(* get pointer to axis data *)
pAxisData := gpAx[nHliAxIdx];
IF pAxisData^.ipo_state.cnc_channel_r = nChan THEN (* it's an axis of the channel *)
	(* is a reset commanded *)
	IF pAxisData^.ipo_lc_control.plc_reset.command_r = TRUE THEN
		(* quit this reset *)
		pAxisData^.ipo_lc_control.plc_reset.state_w := TRUE;

		ADSLOG2(strMsg:='Reset of axis: %d', nUDINT:=nAxisNr, strArg:='');

		HLI_AxisReset := TRUE;
	END_IF
END_IF

END_FUNCTION

// ---- POUs/CNC/F6 BlockSearch/HLI_ChannelBlockSearch.TcPOU
FUNCTION_BLOCK HLI_ChannelBlockSearch
VAR_INPUT
	nChan						: UDINT;			(* Number of channel *)
	(* interface values *)
	BlockSearch				: ST_BlockSearch;
END_VAR
VAR_IN_OUT
	bStartWrite				: BOOL;			(* Edge signal *)
	bStartRead				: BOOL;			(* Edge signal *)
END_VAR
VAR_OUTPUT
	Busy						: BOOL;
	Err						: BOOL;
	nErrorState				: UINT;
	(* interface values *)
	nActType					: INT;
	fActDistance			: LREAL;
	bActAutoReturn			: BOOL;
	nActDeviationMax		: UDINT;
	nActBlockNumber		: DINT;
	nActPass					: DINT;
	nActBlockCount			: DINT;
	(* current values *)
	actualBlockNumber		: DINT := 0;
	actualBlockCount		: DINT := 0;
	actualBlockCount_AferReset : DINT := 0;
	coveredDistance		: DINT;
END_VAR
VAR
	pChannel					: POINTER TO HIGH_LEVEL_INTERFACE_CH;
	nHliChIdx				: UDINT;
	bReadStarted			: BOOL;
	bWriteStarted			: BOOL;
	rtStartRead				: R_TRIG;
	rtStartWrite			: R_TRIG;

	fbWriteType				: FB_BlockSearchWrite;
	fbReadType				: FB_BlockSearchRead;

	fbWriteCovDistance	: FB_BlockSearchWrite;
	fbReadCovDistance		: FB_BlockSearchRead;

	fbWriteAutoReturn		: FB_BlockSearchWrite;
	fbReadAutoReturn		: FB_BlockSearchRead;

	fbWriteDeviationMax	: FB_BlockSearchWrite;
	fbReadDeviationMax	: FB_BlockSearchRead;

	fbWriteBlockNumber	: FB_BlockSearchWrite;
	fbReadBlockNumber		: FB_BlockSearchRead;
	fbReadActBlockNumber	: FB_BlockSearchRead;

	fbWriteBlockCount		: FB_BlockSearchWrite;
	fbReadBlockCount		: FB_BlockSearchRead;
	fbReadActBlockCount	: FB_BlockSearchRead;

	fbWritePass				: FB_BlockSearchWrite;
	fbReadPass				: FB_BlockSearchRead;

	nIdxGrp					: UDINT;
	fDist						: LREAL;
	timer1					: TON;				(* Timer to read actual values cyclically *)
	bStartReadAct			: BOOL;

	channelMode 			: DWORD;
	blockSearchStart		: BOOL;
END_VAR

(* ========================================================= *)
(*    FUN: HLI_ChannelBlockSearch                            *)
(* --------------------------------------------------------- *)
(*   Desc:                                                   *)
(* Author: MK                                                *)
(*   Date: 21.12.2011                                        *)
(*   Rev.: 1.0                                               *)
(* ========================================================= *)


nHliChIdx := nChan - 1;

IF nChan <= 0 OR gNrCh < nChan OR			(* check for channel no *)
	gpCh[nHliChIdx] = 0 THEN					(* check for zero pointer *)
	Err := TRUE;
	RETURN; (* e x i t *)
END_IF


pChannel := gpCh[nHliChIdx];
Err := FALSE;
nIdxGrp := 16#00020100 + nChan;
blockSearchStart := FALSE;


(* ----------------------------------- *)
(* --- write block search commands --- *)
(* ----------------------------------- *)

rtStartWrite(CLK:=bStartWrite);
IF rtStartWrite.Q THEN
	bWriteStarted := TRUE;
	bStartWrite := FALSE; (* reset the HMI signal *)
END_IF

IF bWriteStarted THEN
	Busy := TRUE;
	IF BlockSearch.nType = 5 THEN
		BlockSearch.nType := 3;								(* start position by block count *)

		BlockSearch.bAutoReturn := TRUE;
		(*nPass	:= 1;*)
	END_IF

	(* write block search data to Cnc *)
	fDist := BlockSearch.fDistance * 10.0;
	fbWriteType(nIdxGrp:=nIdxGrp, nIdxOffs:=16#49, nLen:=2, bStart:=rtStartWrite.Q, pDest:=ADR(BlockSearch.nType));
	fbWriteCovDistance(nIdxGrp:=nIdxGrp, nIdxOffs:=16#4A, nLen:=8, bStart:=rtStartWrite.Q, pDest:=ADR(fDist));
	fbWriteAutoReturn(nIdxGrp:=nIdxGrp, nIdxOffs:=16#4B, nLen:=1, bStart:=rtStartWrite.Q, pDest:=ADR(BlockSearch.bAutoReturn));
	fbWriteDeviationMax(nIdxGrp:=nIdxGrp, nIdxOffs:=16#4C, nLen:=4, bStart:=rtStartWrite.Q, pDest:=ADR(BlockSearch.nDeviationMax));
	fbWritePass(nIdxGrp:=nIdxGrp, nIdxOffs:=16#60, nLen:=4, bStart:=rtStartWrite.Q, pDest:=ADR(BlockSearch.nPass));

	CASE BlockSearch.nType OF		(* count and number share a part of the memory *)
		3:	fbWriteBlockCount(nIdxGrp:=nIdxGrp, nIdxOffs:=16#5E, nLen:=4, bStart:=rtStartWrite.Q, pDest:=ADR(BlockSearch.nBlockCount));
		4:	fbWriteBlockNumber(nIdxGrp:=nIdxGrp, nIdxOffs:=16#5F, nLen:=4, bStart:=rtStartWrite.Q, pDest:=ADR(BlockSearch.nBlockNumber));
	END_CASE

	IF fbWriteType.Busy = FALSE
		AND fbWriteCovDistance.BUSY = FALSE
		AND fbWriteAutoReturn.BUSY = FALSE
		AND fbWriteDeviationMax.BUSY = FALSE
		AND fbWriteBlockNumber.BUSY = FALSE
		AND fbWritePass.BUSY = FALSE
		AND fbWriteBlockCount.BUSY = FALSE
	THEN
		Busy := FALSE;
		bWriteStarted := FALSE;
		blockSearchStart := TRUE;
	END_IF
END_IF


(* Start block search *)
(*
IF (blockSearchStart) AND ((nType = 3) OR (nType = 4)) THEN
	PLCMachineMode[nChan].Start := TRUE;
END_IF
*)

(* -------------------------------- *)
(* --- read block search states --- *)
(* -------------------------------- *)

rtStartRead(CLK:=bStartRead);
(*rtStartRead(CLK:=Timer.Q);*)
IF rtStartRead.Q THEN
	bReadStarted := TRUE;
END_IF

IF bReadStarted THEN
	Busy := TRUE;

	fbReadType(nIdxGrp:=nIdxGrp, nIdxOffs:=16#61, nLen:=2, bStart:=rtStartRead.Q, pDest:=ADR(nActType));
	fbReadCovDistance(nIdxGrp:=nIdxGrp, nIdxOffs:=16#62, nLen:=8, bStart:=rtStartRead.Q, pDest:=ADR(fActDistance));
	fbReadAutoReturn(nIdxGrp:=nIdxGrp, nIdxOffs:=16#63, nLen:=1, bStart:=rtStartRead.Q, pDest:=ADR(bActAutoReturn));
	fbReadDeviationMax(nIdxGrp:=nIdxGrp, nIdxOffs:=16#64, nLen:=4, bStart:=rtStartRead.Q, pDest:=ADR(nActDeviationMax));
	CASE nActType OF			(* count and number cannot be read within a single cycle! *)
		3: fbReadBlockCount(nIdxGrp:=nIdxGrp, nIdxOffs:=16#76, nLen:=4, bStart:=rtStartRead.Q, pDest:=ADR(nActBlockCount));
		4: fbReadBlockNumber(nIdxGrp:=nIdxGrp, nIdxOffs:=16#77, nLen:=4, bStart:=rtStartRead.Q, pDest:=ADR(nActBlockNumber));
	END_CASE;
	fbReadPass(nIdxGrp:=nIdxGrp, nIdxOffs:=16#78, nLen:=4, bStart:=rtStartRead.Q, pDest:=ADR(nActPass));

	(*
	fbReadActBlockNumber(nIdxGrp:=nIdxGrp, bStart:=rtStartRead.Q, pDest:=ADR(actualBlockNumber));
	fbReadActBlockCount(nIdxGrp:=nIdxGrp, bStart:=rtStartRead.Q, pDest:=ADR(actualBlockCount));
	*)

	IF fbReadType.Busy = FALSE
		AND fbReadCovDistance.Busy = FALSE
		AND fbReadAutoReturn.Busy = FALSE
		AND fbReadDeviationMax.Busy = FALSE
		AND fbReadBlockNumber.Busy = FALSE
		AND fbReadPass.Busy = FALSE
		AND fbReadActBlockNumber.Busy = FALSE
		AND fbReadActBlockCount.Busy = FALSE
	THEN
		Busy := FALSE;

		bReadStarted := FALSE;
		bStartRead := FALSE; (* reset the HMI signal *)
	END_IF
END_IF


(* Start a cyclic timer with period 100 ms *)
timer1(IN := NOT(timer1.Q), PT := T#100MS);
IF timer1.Q THEN
	bStartReadAct := TRUE;
END_IF

IF bStartReadAct THEN
	fbReadActBlockNumber(nIdxGrp:=nIdxGrp, nIdxOffs:=16#0E, nLen:=4, bStart:=TRUE, pDest:=ADR(actualBlockNumber));
	fbReadActBlockCount(nIdxGrp:=nIdxGrp, nIdxOffs:=16#0D, nLen:=4, bStart:=TRUE, pDest:=ADR(actualBlockCount));
	
	IF fbReadActBlockNumber.Busy = FALSE
		AND fbReadActBlockNumber.Busy = FALSE
	THEN
		bStartReadAct := FALSE;
	END_IF
END_IF


(* just read actual covered distance *)
coveredDistance := pChannel^.bahn_state.covered_distance_r;

(* save all the information from the Cnc break *)
channelMode := HLI_ChannelGetMode(nChan);
IF (actualBlockCount <> 0) AND (channelMode = HLI_IMCM_AUTOMATIC_MODE) THEN
	(* Information stayes after reset *)
	actualBlockCount_AferReset := actualBlockCount;
END_IF


(*actualBlockNumber := pglAx[0]^.lr_state.block_nr_r;  asume first axis is always moved *)


(* handshake during block search on/off *)
pChannel^.bahn_lc_control.block_search.enable_w := TRUE;

IF pChannel^.bahn_lc_control.block_search.command_r <>
	pChannel^.bahn_lc_control.block_search.state_w THEN

	(* acknowledge *)
	pChannel^.bahn_lc_control.block_search.state_w := pChannel^.bahn_lc_control.block_search.command_r;

(*
	(* pup up of change *)
	IF pChannel^.bahn_lc_control.block_search.state_w THEN
		ADSLOGDINT( msgCtrlMask := ADSLOG_MSGTYPE_MSGBOX OR ADSLOG_MSGTYPE_LOG,
						msgFmtStr := 'block search: %d', dintArg := 1);
	ELSE
		ADSLOGDINT( msgCtrlMask := ADSLOG_MSGTYPE_MSGBOX OR ADSLOG_MSGTYPE_LOG,
						msgFmtStr := 'block search: %d', dintArg := 0);
	END_IF
*)
END_IF

END_FUNCTION_BLOCK

// ---- POUs/CNC/F6 BlockSearch/FB_BlockSearchWrite.TcPOU
FUNCTION_BLOCK FB_BlockSearchWrite
VAR_INPUT
	nIdxGrp					: UDINT;
	nIdxOffs					: UDINT;
	nLen						: UDINT;
	bStart					: BOOL;
	pDest						: POINTER TO DWORD;
END_VAR
VAR_OUTPUT
	Busy						: BOOL;
	bErr						: BOOL;
END_VAR
VAR
   fbWrite              : ADSWRITE;
   bStarted             : BOOL;
END_VAR

IF bStarted = FALSE THEN
   IF bStart = TRUE THEN
      bStarted := TRUE;
      bErr := FALSE;
      Busy := TRUE;
   END_IF
END_IF

IF bStarted THEN
   (* raising edge of Timer triggers write request *)
   fbWrite(NetID:='', Port:=553, IdxGrp:=nIdxGrp, IdxOffs:=nIdxOffs,
         LEN:=nLen, SrcAddr:=pDest, WRITE:=bStarted, TMOUT:=T#1S);
   IF NOT fbWrite.Busy THEN
      (* There was an error in the execution of the write request *)
      IF fbWrite.Err THEN
         bErr := TRUE;
      END_IF
      fbWrite(WRITE := FALSE);    (* reset because of edge detection in FB ADSWRITE *)
      bStarted := FALSE;
      Busy := FALSE;
   END_IF
END_IF

END_FUNCTION_BLOCK

// ---- POUs/CNC/F6 BlockSearch/FB_BlockSearchRead.TcPOU
FUNCTION_BLOCK FB_BlockSearchRead
VAR_INPUT
	nIdxGrp					: UDINT;
	nIdxOffs					: UDINT;
	nLen						: UDINT;
	bStart					: BOOL;
	pDest						: POINTER TO DWORD;
END_VAR
VAR_OUTPUT
	Busy						: BOOL;
	bErr						: BOOL;
END_VAR
VAR
	fbRead					: ADSREAD;
	bStarted					: BOOL;
END_VAR

IF bStarted = FALSE THEN
	IF bStart = TRUE THEN
		bStarted := TRUE;
		bErr := FALSE;
		Busy := TRUE;
	END_IF
END_IF

IF bStarted THEN
	(* raising edge of Timer triggers read request *)
	fbRead(NetID:='', Port:=553, IdxGrp:=nIdxGrp, IdxOffs:=nIdxOffs,
		LEN:=nLen, DestAddr:=pDest, READ:=bStarted, TMOUT:=T#1S);
	IF NOT fbRead.Busy THEN
		(* There was an error in the execution of the read request *)
		IF fbRead.Err THEN
			bErr := TRUE;
		END_IF
		fbRead(READ := FALSE);    (* reset because of edge detection in FB ADSREAD *)
		bStarted := FALSE;
		Busy := FALSE;
	END_IF
END_IF

END_FUNCTION_BLOCK

// ---- POUs/CNC/F3_Control/HLI_ChannelGetMessage.TcPOU
FUNCTION_BLOCK HLI_ChannelGetMessage
VAR_INPUT
	nChan			: UINT;			(* Number of channel *)
	bExecute  	: BOOL := FALSE;
	bShowDlg		: BOOL := FALSE;
END_VAR
VAR_OUTPUT
	strToPLC		: STRING(HLI_MSG_CONTENT_STRL) := '';
	iMsgType		: DWORD := 0;
END_VAR
VAR
	nHliChIdx	: UINT;
	pChannel		: POINTER TO HIGH_LEVEL_INTERFACE_CH;
	pMsgCU		: POINTER TO MC_CONTROL_MSG_UNIT;
	pMsgToPLC	: POINTER TO STRING(HLI_MSG_CONTENT_STRL);
END_VAR

(* ========================================================= *)
(*     FB: HLI_ChannelGetMessage                             *)
(* --------------------------------------------------------- *)
(*   Desc: Get message from the CNC                          *)
(*   Author: MK                                              *)
(*   Date: 16.11.2006                                        *)
(*   Rev.: 1.00                                              *)
(* ========================================================= *)


nHliChIdx := nChan - 1;

IF nChan <= 0 OR gNrCh < nChan OR			(* check for channel no *)
	gpCh[nHliChIdx] = 0 THEN					(* check for zero pointer *)
	RETURN; (* e x i t *)
END_IF

IF bExecute = FALSE THEN
	RETURN; (* e x i t *)
END_IF

(* Get pointer to data of a specific channel at the HLI *)
pChannel := gpCh[nHliChIdx];

(* Control unit at the HLI that handles channel specific messages *)
pMsgCU := ADR(pChannel^.msg_mc_control);

(* Is the complete message in the control unit? *)
IF pMsgCU^.request_semaphor_rw = TRUE THEN
	(* Pointer to content of the message sent to the PLC *)
	pMsgToPLC := ADR(pMsgCU^.request_r.inhalt);

	(* Get the message from the control unit *)
	strToPLC := pMsgToPLC^;

	CncSystem.Channel[nChan].Message := strToPLC;
	
	(* Get the message type *)
	iMsgType := pMsgCU^.request_r.typ;

	(* Pop up dialog with the message send to the PLC *)
	IF bShowDlg THEN
		ADSLOGSTR( msgCtrlMask :=ADSLOG_MSGTYPE_MSGBOX OR ADSLOG_MSGTYPE_LOG,
						msgFmtStr := 'Message sent to PLC via HLI:%s',
						strArg := strToPLC);
	END_IF

	(* Acknowledge that you got the message *)
	pChannel^.msg_mc_control.request_semaphor_rw  := FALSE;
END_IF

END_FUNCTION_BLOCK

// ---- POUs/CncAxisEnable.TcPOU
PROGRAM CncAxisEnable
VAR_INPUT
	bEnable					: BOOL;
END_VAR
VAR
	bTorquePermission		: BOOL;
	bFeedhold				: BOOL;
	bDriveOn					: BOOL;

	T_DriveOn				: TON;
END_VAR

(* ========================================================= *)
(*    PRG: CncAxisEnable                                     *)
(* --------------------------------------------------------- *)
(*   Desc:                                                   *)
(* Author: MK                                                *)
(*   Date: 21.12.2011                                        *)
(*   Rev.: 1.0                                               *)
(* ========================================================= *)


(* Enable drive, order depends by type of drive and fieldbus *)
T_DriveOn(IN:=bEnable, PT:=T#1S);
IF bEnable THEN
	bDriveOn			:= TRUE;
	IF T_DriveOn.Q THEN
		bTorquePermission	:= TRUE;
		bFeedhold			:= TRUE;
	END_IF
ELSE
	bTorquePermission	:= FALSE;
	bFeedhold			:= FALSE;
	bDriveOn				:= FALSE;
END_IF

(* Enable drive, order depends by type of drive and fieldbus *)
(*
T_DriveOn(IN:=bEnable, PT:=T#1s);
IF bEnable THEN
	bTorquePermission	:= TRUE;
	bFeedhold			:= TRUE;
	IF T_DriveOn.Q THEN
		bDriveOn			:= TRUE;
	END_IF
ELSE
	bTorquePermission	:= FALSE;
	bFeedhold			:= FALSE;
	bDriveOn				:= FALSE;
END_IF
*)


(* Controller Enable, axis specific *)
HLI_AxisSetFeedHold(Axis:=1, TorquePermission:=bTorquePermission, Feedhold:=bFeedhold, DriveOn:=bDriveOn);
HLI_AxisSetFeedHold(Axis:=2, TorquePermission:=bTorquePermission, Feedhold:=bFeedhold, DriveOn:=bDriveOn);
HLI_AxisSetFeedHold(Axis:=3, TorquePermission:=bTorquePermission, Feedhold:=bFeedhold, DriveOn:=bDriveOn);
HLI_AxisSetFeedHold(Axis:=4, TorquePermission:=bTorquePermission, Feedhold:=bFeedhold, DriveOn:=bDriveOn);
HLI_AxisSetFeedHold(Axis:=5, TorquePermission:=bTorquePermission, Feedhold:=bFeedhold, DriveOn:=bDriveOn);

HLI_AxisSetFeedHold(Axis:=6, TorquePermission:=bTorquePermission, Feedhold:=bFeedhold, DriveOn:=bDriveOn);
HLI_AxisSetFeedHold(Axis:=7, TorquePermission:=bTorquePermission, Feedhold:=bFeedhold, DriveOn:=bDriveOn);
HLI_AxisSetFeedHold(Axis:=8, TorquePermission:=bTorquePermission, Feedhold:=bFeedhold, DriveOn:=bDriveOn);

END_PROGRAM

// ---- POUs/CNC/F3_Control/HLI_AxisSetFeedHold.TcPOU
FUNCTION HLI_AxisSetFeedHold : BOOL
VAR_INPUT
	Axis					: UDINT;
	TorquePermission	: BOOL;
	Feedhold				: BOOL;
	DriveOn				: BOOL;
END_VAR
VAR
	nHliAxIdx			: UDINT;		(* Index of axis specific HLI area *)
END_VAR

(* ========================================================= *)
(*    FUN: HLI_AxisSetFeedHold                               *)
(* --------------------------------------------------------- *)
(*   Desc:                                                   *)
(* Author: MK                                                *)
(*   Date: 21.12.2011                                        *)
(*   Rev.: 1.0                                               *)
(* ========================================================= *)


nHliAxIdx := Axis - 1;

IF Axis < 1	OR gNrAx < Axis			(* check for axis no *)
	OR gpAx[nHliAxIdx] = 0 THEN		(* check for zero pointer *)
	HLI_AxisSetFeedHold := FALSE;
	RETURN; (* e x i t *)
END_IF

(* set regulation and feed *)
gpAx[nHliAxIdx]^.lr_mc_control.torque_permission.command_w := TorquePermission;
gpAx[nHliAxIdx]^.lr_mc_control.release_feedhold.command_w := Feedhold;
gpAx[nHliAxIdx]^.lr_mc_control.drive_on.command_w := DriveOn;

HLI_AxisSetFeedHold := TRUE;

END_FUNCTION

// ---- POUs/CNC/F3_Control/HLI_AxisSetTrackingOperation.TcPOU
FUNCTION HLI_AxisSetTrackingOperation : BOOL
VAR_INPUT
	nAxisNr				: UDINT;
	bPLCAxisEnable    : BOOL;
END_VAR
VAR
	nHliAxIdx			: UDINT;		(* Index of axis specific HLI area *)
END_VAR

(* ========================================================= *)
(*    FUN: HLI_AxisSetTrackingOperation                      *)
(* --------------------------------------------------------- *)
(*   Desc:                                                   *)
(*   Author: TV                                              *)
(*   Date: 21.12.2012                                        *)
(*   Rev.: 1.0                                               *)
(* ========================================================= *)


nHliAxIdx := nAxisNr - 1;

IF nAxisNr < 1	OR gNrAx < nAxisNr	(* check for axis no *)
	OR gpAx[nHliAxIdx] = 0 THEN		(* check for zero pointer *)
	HLI_AxisSetTrackingOperation := FALSE;
	RETURN; (* e x i t *)
END_IF


(* The axis is set to tracking operation (follow up) on or off, i.e. the control loop is opened.
   The command position implicitly is set to the actual position. *)
IF gpAx[nHliAxIdx]^.lr_state.axis_state_r = HLI_AXIS_ERROR OR NOT bPLCAxisEnable THEN
	gpAx[nHliAxIdx]^.lr_mc_control.follow_up.command_w := TRUE;
	HLI_AxisSetTrackingOperation := TRUE;
ELSE
	gpAx[nHliAxIdx]^.lr_mc_control.follow_up.command_w := FALSE;
	HLI_AxisSetTrackingOperation := FALSE;
END_IF

END_FUNCTION

// ---- POUs/CNC/F3_Control/HLI_AxisSetReferenceCam.TcPOU
FUNCTION HLI_AxisSetReferenceCam : BOOL
VAR_INPUT
	Axis					: UDINT;
	bReferenceCam		: BOOL;
END_VAR
VAR
	nHliAxIdx			: UDINT;		(* Index of axis specific HLI area *)
END_VAR

(* ========================================================= *)
(*    FUN: HLI_AxisSetReferenceCam                           *)
(* --------------------------------------------------------- *)
(*   Desc:                                                   *)
(* Author: MK                                                *)
(*   Date: 21.12.2011                                        *)
(*   Rev.: 1.0                                               *)
(* ========================================================= *)


nHliAxIdx := Axis - 1;

IF Axis < 1	OR gNrAx < Axis				(* check for axis no *)
	OR gpAx[nHliAxIdx] = 0 THEN			(* check for zero pointer *)
	HLI_AxisSetReferenceCam := FALSE;
	RETURN; (* e x i t *)
END_IF

(* set reference cam *)
gpAx[nHliAxIdx]^.lr_mc_control.reference_cam.command_w := bReferenceCam;

HLI_AxisSetReferenceCam := TRUE;

END_FUNCTION

// ---- POUs/CNC/F3_Control/HLI_ChannelSetOverride.TcPOU
FUNCTION HLI_ChannelSetOverride : BOOL
VAR_INPUT
	nChan					: UINT;			(* Number of channel *)
	nOverride			: UINT;
END_VAR
VAR
	nHliChIdx			: UINT;
END_VAR

(* ========================================================= *)
(*    FUN: HLI_ChannelSetOverride                            *)
(* --------------------------------------------------------- *)
(*   Desc: Set the channel Override                          *)
(* Author: MK                                                *)
(*   Date: 21.12.2011                                        *)
(*   Rev.: 1.0                                               *)
(* ========================================================= *)


nHliChIdx := nChan - 1;

IF nChan <= 0 OR gNrCh < nChan OR			(* check for channel no *)
	gpCh[nHliChIdx] = 0 THEN					(* check for zero pointer *)
	HLI_ChannelSetOverride := FALSE;
	RETURN; (* e x i t *)
END_IF

(* Limit the override *)
IF nOverride > 1200	THEN nOverride := 1200; END_IF
IF nOverride < 0 THEN nOverride := 0; END_IF

gpCh[nHliChIdx]^.bahn_mc_control.override_feedrate.command_w := nOverride;

HLI_ChannelSetOverride := TRUE;

END_FUNCTION

// ---- POUs/CNC/F3_Control/HLI_ChannelSetSuspendAxisOutput.TcPOU
FUNCTION HLI_ChannelSetSuspendAxisOutput : BOOL
VAR_INPUT
	nChan					: UDINT;			(* Number of channel *)
	bSuspendAxis		: BOOL;
END_VAR
VAR
	nHliChIdx			: UDINT;
END_VAR

(* ========================================================= *)
(*    FUN: HLI_ChannelSuspendAxisOutput                      *)
(* --------------------------------------------------------- *)
(*   Desc:                                                   *)
(* Author: MK                                                *)
(*   Date: 18.04.2003                                        *)
(*   Rev.: 1.0                                               *)
(* ========================================================= *)


nHliChIdx := nChan - 1;

IF nChan <= 0 OR gNrCh < nChan OR			(* check for channel no *)
	gpCh[nHliChIdx] = 0 THEN					(* check for zero pointer *)
	HLI_ChannelSetSuspendAxisOutput := FALSE;
	RETURN; (* e x i t *)
END_IF

gpCh[nHliChIdx]^.bahn_mc_control.suspend_axis_output.command_w := bSuspendAxis;

HLI_ChannelSetSuspendAxisOutput := TRUE;

END_FUNCTION

// ---- POUs/CNC/F9_Misc/HandWheel/PRG_ManualModeG201.TcPOU
PROGRAM PRG_ManualModeG201
VAR_INPUT
	nChan						: UDINT;		(* starts with 1, 2,... *)
END_VAR
VAR
	nAxis						: UINT := 3;	(* X=1; Y=2; Z=3 *)
	bOpModeAuto				: BOOL;		(* activates, deactivates operation *) 
	bManualIsOn				: BOOL;
	bEndOfManualMode		: BOOL;
	bManualModeErr			: BOOL;		(* inicates error *)

	AxisManualModeG201	: HLI_AxisManualMode;
	manualModeParam		: ST_ManualModeParam;
	pChannel					: POINTER TO HIGH_LEVEL_INTERFACE_CH;  		
	nHliChIdx				: UDINT;
	fbRTrig					: R_TRIG;
	fbFTrig					: F_TRIG;
	hbStateAxis				: DINT;
END_VAR

(* ========================================================= *)
(*    PRG: PRG_ManualModeG201                                *)
(* --------------------------------------------------------- *)
(*   Desc: Axis manual mode with parallel interpolation G201 *)
(* Author: MK                                                *)
(*   Date: 12.05.2016                                        *)
(*   Rev.: 1.0                                               *)
(* ========================================================= *)


nHliChIdx := nChan - 1;

IF nChan <= 0 OR gNrCh < nChan OR			(* check for channel no *)
	gpCh[nHliChIdx] = 0 THEN					(* check for zero pointer *)
	RETURN; (* e x i t *)
END_IF

(* axis number must be 1, 2, 3,... *)
IF nAxis < 1 THEN
	RETURN;
END_IF

(* activates operation only in automatic mode *)
bOpModeAuto := (HLI_ChannelGetMode(nChan:=nChan) = HLI_IMCM_AUTOMATIC_MODE);

(* This enables automatically the axis manual movement *)
pChannel := gpCh[nHliChIdx];
hbStateAxis := pChannel^.bahn_state.coord_r[nAxis - 1].hb_display_r.state;	(* Status of the axis | 0=Inactive, 1=Ready, 2=Active *)

fbRTrig(CLK := (hbStateAxis<>0) AND bOpModeAuto);
fbFTrig(CLK := (hbStateAxis<>0) AND bOpModeAuto);

IF fbRTrig.Q OR bManualIsOn THEN
	IF fbRTrig.Q THEN			(* activation *)
		bManualIsOn := TRUE;
		bEndOfManualMode := FALSE;
	ELSIF fbFTrig.Q THEN		(* deactivation *)
		bEndOfManualMode := TRUE;
	END_IF
	
	manualModeParam.nOpMode := UDINT_TO_UINT(HLI_HB_MODE_HR);
	manualModeParam.nLogAxisNr := nAxis;		// PlcManualModeSelectedAxis;
	manualModeParam.nControlElement := 1;
	manualModeParam.nHandwheelNr := 0;
	manualModeParam.nHandwheelIncs := PlcManualModeHandWheelIncs;
	manualModeParam.nHandwheelRes := PlcManualModeHandWheelRes; 
	manualModeParam.nTipSpeed := PlcManualModeSpeed;
	manualModeParam.nJogSpeed := PlcManualModeSpeed;
	manualModeParam.nJogDistance := PlcManualModeIncrements;

	(* manual mode keypress *)
	manualModeParam.bKeyPos := PlcManualModeRightKey;
	manualModeParam.bKeyNeg := PlcManualModeLeftKey;
	manualModeParam.bKeyRapid := PlcManualModeRapidFeedKey;

	
	AxisManualModeG201(nChan			:= nChan,
							sProgramName	:= '',
							bEndManual		:= bEndOfManualMode,
							ManualModeParam:= manualModeParam, 
							nKeyUnitIdx		:= 0,
							bManualModeHMI	:= FALSE,
							bReset			:= FALSE,
							bG201				:= TRUE);
							
	IF AxisManualModeG201.Busy = FALSE THEN
		AxisManualModeG201.bG201 := FALSE;
		bEndOfManualMode := FALSE;
		bManualIsOn := FALSE;
	END_IF
	bManualModeErr := AxisManualModeG201.Err;
END_IF

END_PROGRAM

// ---- POUs/CncMFunctions.TcPOU
PROGRAM CncMFunctions
VAR

END_VAR

(* ========================================================= *)
(*    FUN: CncMFunctions                                     *)
(* --------------------------------------------------------- *)
(*   Desc:                                                   *)
(* Author: MK                                                *)
(*   Date: 21.12.2011                                        *)
(*   Rev.: 1.0                                               *)
(* ========================================================= *)

(*
IF CncSystem.Channel[1].M[40] = TRUE THEN
	CncSystem.Channel[1].M[40] := FALSE;
END_IF
*)

(* M-functions *)
IF CNCSystem.Channel[1].M[17] = TRUE THEN
	CNCSystem.Channel[1].M[17] := FALSE;
END_IF

(*IF CNCSystem.Channel[1].M[52] = TRUE THEN
	Temp_Tabuleiro_set:=CNCSystem.Channel[1].M_Argument[52];
		IF (IOs.Temp_Tabuleiro<Temp_Tabuleiro_set+100 AND IOs.Temp_Tabuleiro>Temp_Tabuleiro_set-100) OR Temp_Tabuleiro_set=0 THEN
			CNCSystem.Channel[1].M[52] := FALSE;
		END_IF
END_IF*)

END_PROGRAM

// ---- POUs/CncPlcManualFunctions.TcPOU
PROGRAM CncPlcManualFunctions
VAR
	bSetString					: BOOL := TRUE;
	PLCManual_Off				: BYTE := 0;
	PLCManual_StatusLeft		: BYTE := 1;
	PLCManual_StatusRight	: BYTE := 2;
	PLCManual_LockLeft		: BYTE := 32;
	PLCManual_LockRight		: BYTE := 64;
END_VAR

(* ========================================================= *)
(*    FUN: CncPlcManualFunctions                             *)
(* --------------------------------------------------------- *)
(*   Desc:                                                   *)
(* Author: MK                                                *)
(*   Date: 21.08.2008                                        *)
(*   Rev.: 1.0                                               *)
(* ========================================================= *)


(* Manual functions *)
PortalStatus[1] := PLCManual_StatusLeft;
PortalStatus[2] := PLCManual_StatusLeft;
PortalStatus[3] := PLCManual_StatusLeft;
PortalStatus[4] := PLCManual_LockRight;

SchweissenStatus[1] := PLCManual_Off;
SchweissenStatus[2] := PLCManual_StatusLeft;
SchweissenStatus[3] := PLCManual_StatusRight;
SchweissenStatus[4] := PLCManual_StatusLeft;

MSGList3[3] := PortalOn[7];


IF bSetString THEN
	PortalActValueLeft[3] := INT_TO_STRING(DemoUpDown.UpDown);
	PortalActValueLeft[4] := INT_TO_STRING(DemoUpDown.UpDown);
	PortalActValueLeft[5] := INT_TO_STRING(DemoUpDown.UpDown);
END_IF

END_PROGRAM

// ---- POUs/CncPlcMessages.TcPOU
PROGRAM CncPlcMessages
VAR
	bShowMessage		: BOOL;
	
	event1				: FB_SimpleAdsLogEvent;
	event2				: FB_SimpleAdsLogEvent;
	bStartEvent			: BOOL;
	bStartEvent2		: BOOL;
	i						: INT;
END_VAR

(* ========================================================= *)
(*    FUN: CncPlcMessages                                    *)
(* --------------------------------------------------------- *)
(*   Desc:                                                   *)
(* Author: MK                                                *)
(*   Date: 21.12.2011                                        *)
(*   Rev.: 1.0                                               *)
(* ========================================================= *)


(* Messages *)
MSGList1[5] := bShowMessage;
MSGList1[6] := bShowMessage;
MSGList1[7] := bShowMessage;

(*FOR i:=1 TO 50 DO
	MSGList2[i] := bShowMessage;
END_FOR*)


// Eventlogger
(*
event1(SourceID:=50, EventID:=3, bSetEvent:=bStartEvent);
errId := event1.ErrId;

event2(SourceID:=50, EventID:=4, bSetEvent:=bStartEvent2);
*)

END_PROGRAM

// ---- POUs/CncRefPosOffs.TcPOU
PROGRAM CncRefPosOffs
VAR
END_VAR

(* ========================================================= *)
(*    FUN: CncRefPosOffs                                     *)
(* --------------------------------------------------------- *)
(*   Desc:                                                   *)
(* Author: MK                                                *)
(*   Date: 21.12.2011                                        *)
(*   Rev.: 1.0                                               *)
(* ========================================================= *)


gpAx[0]^.lr_mc_control.refpos_position.enable_w := TRUE;
gpAx[1]^.lr_mc_control.refpos_position.enable_w := TRUE;
gpAx[2]^.lr_mc_control.refpos_position.enable_w := TRUE;

gpAx[0]^.lr_mc_control.set_reference_position.enable_w := TRUE;  
gpAx[1]^.lr_mc_control.set_reference_position.enable_w := TRUE;  
gpAx[2]^.lr_mc_control.set_reference_position.enable_w := TRUE;  



gpAx[0]^.lr_mc_control.refpos_position.command_w := 100 * 10000;
gpAx[1]^.lr_mc_control.refpos_position.command_w := 200 * 10000;
gpAx[2]^.lr_mc_control.refpos_position.command_w := 300 * 10000;

gpAx[0]^.lr_mc_control.set_reference_position.command_w := TRUE;  
gpAx[1]^.lr_mc_control.set_reference_position.command_w := TRUE;  
gpAx[2]^.lr_mc_control.set_reference_position.command_w := TRUE;

END_PROGRAM

// ---- POUs/CncVariables.TcPOU
PROGRAM CncVariables
VAR_INPUT
END_VAR
VAR
	VE						: ST_VEVariableConfig;
	v1 : DINT;
	v4 : DINT;
	v5 : DINT;
END_VAR

(* ========================================================= *)
(*    PRG: CncVariables                                      *)
(* --------------------------------------------------------- *)
(*   Desc:                                                   *)
(* Author: MK                                                *)
(*   Date: 21.12.2011                                        *)
(*   Rev.: 1.0                                               *)
(* ========================================================= *)



(* External Variables in the CNC, must be set only at startup *)
VE.VARIABLE_1 := LinkVEChannelStructure(nChan:=1, nVEIndex:=0, bGlobal:=TRUE);
VE.VARIABLE_4 := LinkVEChannelStructure(nChan:=1, nVEIndex:=3, bGlobal:=TRUE);
VE.VARIABLE_5 := LinkVEChannelStructure(nChan:=1, nVEIndex:=4, bGlobal:=TRUE);


v1 := VE.VARIABLE_1^[0];
v4 := VE.VARIABLE_4^;
v5 := VE.VARIABLE_5^;

(*
VE.VARIABLE_1^[0] := 300;
VE.VARIABLE_1^[1] := 1234;
*)

(*
VE.VARIABLE_1^[0] := 100;
VE.VARIABLE_1^[1] := 200;
VE.VARIABLE_1^[2] := 300;
VE.VARIABLE_1^[3] := 400;
VE.VARIABLE_4^ := 500;
*)

END_PROGRAM

// ---- POUs/CNC/F5_Variables/LinkVEChannelStructure.TcPOU
FUNCTION LinkVEChannelStructure : POINTER TO DWORD
VAR_INPUT
	nChan				: INT;			(* Number of Channel 1...nChannel *)
	nVEIndex			: DINT;			(* Index of variable  range 1...HLI_VE_VALUEMAX *)
	bGlobal			: BOOL;			(* serves access to the global variable array *)
END_VAR
VAR
	pVeData			: POINTER TO HLI_V_E_DATA := 0;
	ptr      		: POINTER TO DWORD;
END_VAR


IF nVEIndex >= 0 THEN
	IF bGlobal = TRUE  THEN
		(* global cnc variable data *)
		pVeData := gpVEGlobal;
	ELSE
		(* channel specific cnc variable data *)
		IF nChan <= 0 OR nChan < HLI_SYS_CH_MAXIDX THEN
			RETURN;
		END_IF
		pVeData := gpVECh[nChan];
	END_IF

	IF pVeData <> 0 THEN
		ptr := pVeData +  24 * nVEIndex;

		LinkVEChannelStructure := ptr; (* successfully completed return *)
	END_IF
END_IF



(*
pLRealVal : POINTER TO LREAL;
LRealVal : LREAL;
VeOffset : DINT;
VeOffset := (VarNr - 1) * (HLI_EXT_VAR_STR_MAXIDX + 1) / 4 + 1;
pLRealVal := gpVEGlobal^.ext_var32[VeOffset]);
LRealVal := pLRealVal^;
*)

END_FUNCTION

// ---- POUs/Temperature Controller/TController_Enable.TcPOU
PROGRAM TController_Enable
VAR
	
END_VAR

(*Desligar ventoinhas depois de máquina arrefecer *)
IF IOs.Temp_Camara_in<4000 AND IOs.Temp_Camara_out<4000 AND Temp_Camara_set<4000 THEN
	IOs.IO_Out_Vent_Camara:=FALSE;
	IOs.IO_Out_Vent_cabl_X:=FALSE;
	IOs.IO_Out_Vent_Porta:=FALSE;
	IOs.IO_Out_Vent_Quadro1:=FALSE;
END_IF

(* Ligar Recirculação do ar da camara se temperatura for definida ou superior a 50ºC*)
IF IOs.Temp_Camara_in>5000 OR IOs.Temp_Camara_out>5000 OR Temp_Camara_set<>0 OR IOs.A_Out_Aque_Ar<>0 THEN
	IOs.IO_Out_Vent_Camara:=TRUE;
END_IF

(*Ligar refrigeração da mesa se temperatura do tabuleiro superar os 80ºC*)
IF IOs.Temp_Tabuleiro>8000 THEN
	IOs.IO_Out_Vent_cabl_X:=TRUE;
END_IF

(* Ligar refrigeração da câmara só quando a temperatura superar os 50ºC (aquecimento mais rápido)*)
IF IOs.Temp_Camara_out>5000 OR IOs.Temp_Camara_in>5000 THEN
	IOs.IO_Out_Vent_cabl_X:=TRUE;
	IOs.IO_Out_Vent_Porta:=TRUE;
	IOs.IO_Out_Vent_Quadro1:=TRUE;
END_IF

(* Ligar Chiller quando temperatura do extrusor for definida, ou temperatura da câmara acima dos 50ºC. Desligar quando tudo estiver abaixo dos 40ºC*)
IF  Temp_Extrusor_1_set<>0 OR Temp_Camara_set>5000 OR IOs.Temp_Camara_in>5000 OR IOs.Temp_Camara_out>5000 OR IOs.Temp_Extrusor_1>5000 THEN
	IOs.IO_Out_Chiller:=TRUE;
	IOs.IO_Out_Vent_Quadro1:=TRUE;
	ELSIF IOs.Temp_Camara_in<4000 AND IOs.Temp_Camara_out<4000 AND IOs.Temp_Extrusor_1<4000 THEN
 		IOs.IO_Out_Chiller:=FALSE;	
END_IF

(*Ligar segundo set de ventoinhas do quadro se temperatura passar os 35ºC*)
IF IOs.Temp_Quadro>3500 THEN
	IOs.IO_Out_Vent_Quadro2:=TRUE;
	ELSIF IOs.Temp_Quadro<3000 THEN
		IOs.IO_Out_Vent_Quadro2:=FALSE;
END_IF

(*Inicio dos controladores ou desligar saidas*)
IF Temp_Tabuleiro_set<>0 THEN
	PTab();
ELSE
	IOs.IO_Out_Aque_Mesa:=0;
END_IF

IF Temp_Extrusor_1_set<>0 THEN
	Pext();
ELSE
	IOs.IO_Out_Aque_Extrusor:=0;
END_IF

IOs.IO_Out_Chiller:=1;

IF Temp_Camara_set<>0 THEN	
	PCamara();
ELSE 
	IOs.A_Out_Aque_Ar:=0;
END_IF


IF IOs.IO_In_Emergencia=1 THEN
	IOs.A_Out_Aque_Ar:=0;
END_IF

END_PROGRAM

// ---- POUs/Temperature Controller/PTab.TcPOU
PROGRAM PTab

VAR
	fSetpointValue					: FLOAT;
	fActualValue					: FLOAT;
	fManSyncValue					: FLOAT;
	bSync							: BOOL;

	fOut							: FLOAT;
	bHold							: BOOL;

	eMode							: E_CTRL_MODE;
	stCTRL_PID_PARAMS				: ST_CTRL_PID_PARAMS;

	eErrorId						: E_CTRL_ERRORCODES;
	bError							: BOOL;
	bARWactive						: BOOL;

	fbCTRL_PID						: FB_CTRL_PID;

	bInit							: BOOL	:= TRUE;
	fbTON							: TON;
END_VAR

IF bInit
THEN
	(* Init parameter struct *)
	stCTRL_PID_PARAMS.tCtrlCycleTime	:= T#10MS;
	stCTRL_PID_PARAMS.tTaskCycleTime	:= T#10MS;
	stCTRL_PID_PARAMS.fKp				:= 0.15162;			(* proportional gain Kp		*)
	stCTRL_PID_PARAMS.tTn				:= T#1338.57S;		(* integral action time Tn	*)
	stCTRL_PID_PARAMS.tTv				:= T#100S;		(* derivative action time Tv*)
	stCTRL_PID_PARAMS.tTd				:= T#21.9449S;		(* damping time	Td			*)
	stCTRL_PID_PARAMS.fOutMaxLimit		:= 100;			(* maximum output limit		*)
	stCTRL_PID_PARAMS.fOutMinLimit		:= 0;			(* minimum output limit		*)

	(* ACTIVE --> normal operation *)
	eMode								:= eCTRL_MODE_ACTIVE;

	(* Reset init flag *)
	bInit								:= FALSE;
END_IF

	(* Call controller function block *)
fbCTRL_PID(		fSetpointValue			:= Temp_Tabuleiro_set,
					fActualValue		:= IOs.Temp_Tabuleiro,
					fManSyncValue		:= fManSyncValue,
					bSync				:= bSync,
					eMode				:= eMode,
					bHold				:= bHold,
					stParams			:= stCTRL_PID_PARAMS,
					fOut				=> fOut,
					bARWactive			=> bARWactive,
					eErrorId			=> eErrorId,
					bError				=> bError
				);
IF bError=FALSE THEN	
		(* Call PWM function  *)
	PTab_Out(fPwmInput:=fOut);
ELSE
	PTab_Out(fPwmInput:=0);
	(*Escrever o erro para a HMI*)
END_IF

END_PROGRAM

// ---- POUs/Temperature Controller/PTab_Out.TcPOU
PROGRAM PTab_Out

VAR_INPUT
	fPwmInput								: FLOAT;	
END_VAR

VAR
	bPwmOutBitPos							: BOOL;
	bPwmOutBitNeg							: BOOL;

	fbCTRL_PWM_OUT							: FB_CTRL_PWM_OUT;
	stCTRL_PWM_OUT_PARAMS					: ST_CTRL_PWM_OUT_PARAMS;

	eMode									: E_CTRL_MODE;
	eErrorId								: E_CTRL_ERRORCODES;
	bError									: BOOL;

	bInit									: BOOL		:= TRUE;
	fDelta									: FLOAT	:= 0.05;
END_VAR

IF bInit
THEN
	(* Init parameter struct *)
	stCTRL_PWM_OUT_PARAMS.tTaskCycleTime	:= T#10MS;
	stCTRL_PWM_OUT_PARAMS.tPWMPeriod		:= T#200MS;

	(* ACTIVE --> normal operation *)
	eMode									:= eCTRL_MODE_ACTIVE;

	(* Reset the init flag *)
	bInit									:= FALSE;
END_IF

fbCTRL_PWM_OUT(		fPwmInput				:= fPwmInput,
							eMode			:= eMode,
							stParams		:= stCTRL_PWM_OUT_PARAMS,
							
							bPwmOutBitPos	=> bPwmOutBitPos,
							bPwmOutBitNeg	=> bPwmOutBitNeg,
							bError			=> bError,
							eErrorId		=> eErrorId
						);
						
	(* Output sign   *)
IOS.IO_Out_Aque_Mesa:=bPwmOutBitPos;

END_PROGRAM

// ---- POUs/Temperature Controller/PExt.TcPOU
PROGRAM PExt
VAR
	fSetpointValue					: FLOAT		:= 40000;
	fActualValue					: FLOAT;
	fManSyncValue					: FLOAT;
	bSync							: BOOL;

	fOut							: FLOAT;
	bHold							: BOOL;

	eMode							: E_CTRL_MODE;
	stCTRL_PID_PARAMS				: ST_CTRL_PID_PARAMS;

	eErrorId						: E_CTRL_ERRORCODES;
	bError							: BOOL;
	bARWactive						: BOOL;

	fbCTRL_PID						: FB_CTRL_PID;

	bInit							: BOOL	:= TRUE;
	fbTON							: TON;
END_VAR

IF bInit
THEN
	(* Init parameter struct *)
	stCTRL_PID_PARAMS.tCtrlCycleTime	:= T#10MS;
	stCTRL_PID_PARAMS.tTaskCycleTime	:= T#10MS;
	stCTRL_PID_PARAMS.fKp				:= 0.17607;			(* proportional gain Kp		*)
	stCTRL_PID_PARAMS.tTn				:= T#334.9185S;		(* integral action time Tn	*)
	stCTRL_PID_PARAMS.tTv				:= T#50S;		(* derivative action time Tv*)
	stCTRL_PID_PARAMS.tTd				:= T#3.4776S;		(* damping time	Td			*)
	stCTRL_PID_PARAMS.fOutMaxLimit		:= 100;			(* maximum output limit		*)
	stCTRL_PID_PARAMS.fOutMinLimit		:= 0;			(* minimum output limit		*)

	(* ACTIVE --> normal operation *)
	eMode								:= eCTRL_MODE_ACTIVE;

	(* Reset init flag *)
	bInit								:= FALSE;
END_IF

	(* Call controller function block *)
fbCTRL_PID(		fSetpointValue			:= Temp_Extrusor_1_set,
					fActualValue		:= IOS.Temp_Extrusor_1,
					fManSyncValue		:= fManSyncValue,
					bSync				:= bSync,
					eMode				:= eMode,
					bHold				:= bHold,
					stParams			:= stCTRL_PID_PARAMS,
					fOut				=> fOut,
					bARWactive			=> bARWactive,
					eErrorId			=> eErrorId,
					bError				=> bError
			);
IF bError=FALSE THEN			
		(* Call PWM function  *)
	PExt_Out(fPwmInput:=fOut);
ELSE
	PExt_Out(fPwmInput:=0);
	(*Escrever o erro para a HMI*)
END_IF

END_PROGRAM

// ---- POUs/Temperature Controller/PExt_Out.TcPOU
PROGRAM PExt_Out

VAR_INPUT
	fPwmInput								: FLOAT;	
END_VAR

VAR
	bPwmOutBitPos							: BOOL;
	bPwmOutBitNeg							: BOOL;

	fbCTRL_PWM_OUT							: FB_CTRL_PWM_OUT;
	stCTRL_PWM_OUT_PARAMS					: ST_CTRL_PWM_OUT_PARAMS;

	eMode									: E_CTRL_MODE;
	eErrorId								: E_CTRL_ERRORCODES;
	bError									: BOOL;

	bInit									: BOOL	:= TRUE;
	fDelta									: FLOAT	:= 0.05;
	
END_VAR

IF bInit THEN
	(* Init parameter struct *)
	stCTRL_PWM_OUT_PARAMS.tTaskCycleTime	:= T#10ms;
	stCTRL_PWM_OUT_PARAMS.tPWMPeriod		:= T#200Ms;

	(* ACTIVE --> normal operation *)
	eMode									:= eCTRL_MODE_ACTIVE;

	(* Reset init flag *)
	bInit									:= FALSE;
END_IF

	(* Call function block *)
fbCTRL_PWM_OUT(		fPwmInput				:= fPwmInput,
							eMode			:= eMode,
							stParams		:= stCTRL_PWM_OUT_PARAMS,
							
							bPwmOutBitPos	=> bPwmOutBitPos,
							bPwmOutBitNeg	=> bPwmOutBitNeg,
							bError			=> bError,
							eErrorId		=> eErrorId
						);
						
	(* Output sign   *)
IOS.IO_Out_Aque_Extrusor:=bPwmOutBitPos;

END_PROGRAM

// ---- POUs/Temperature Controller/PCamara.TcPOU
PROGRAM PCamara

VAR
	fSetpointValue					: FLOAT		:= 40000;
	fActualValue					: FLOAT;
	fManSyncValue					: FLOAT;
	bSync							: BOOL;

	fOut							: FLOAT;
	bHold							: BOOL;

	eMode							: E_CTRL_MODE;
	stCTRL_PID_PARAMS				: ST_CTRL_PID_PARAMS;

	eErrorId						: E_CTRL_ERRORCODES;
	bError							: BOOL;
	bARWactive						: BOOL;

	fbCTRL_PID						: FB_CTRL_PID;

	bInit							: BOOL	:= TRUE;
	fbTON							: TON;

END_VAR

IF bInit THEN

	(* Init parameter struct *)
	stCTRL_PID_PARAMS.tCtrlCycleTime	:= T#10MS;
	stCTRL_PID_PARAMS.tTaskCycleTime	:= T#10MS;
	stCTRL_PID_PARAMS.fKp				:= 1.0;			(* proportional gain Kp		*)
	stCTRL_PID_PARAMS.tTn				:= T#1S;		(* integral action time Tn	*)
	stCTRL_PID_PARAMS.tTv				:= T#200MS;		(* derivative action time Tv*)
	stCTRL_PID_PARAMS.tTd				:= T#100MS;		(* damping time	Td			*)
	stCTRL_PID_PARAMS.fOutMaxLimit		:= 100;			(* maximum output limit		*)
	stCTRL_PID_PARAMS.fOutMinLimit		:= 0;			(* minimum output limit		*)

	(* ACTIVE --> normal operation *)
	eMode								:= eCTRL_MODE_ACTIVE;

	(* Reset init flag *)
	bInit								:= FALSE;
	
END_IF

	(* Call controller function block *)
fbCTRL_PID(		fSetpointValue			:= Temp_Camara_Set,
					fActualValue		:= IOS.Temp_Camara_out,
					fManSyncValue		:= fManSyncValue,
					bSync				:= bSync,
					eMode				:= eMode,
					bHold				:= bHold,
					stParams			:= stCTRL_PID_PARAMS,
					fOut				=> fOut,
					bARWactive			=> bARWactive,
					eErrorId			=> eErrorId,
					bError				=> bError
			);
	
	(* Call output function only if ventilations is active (avoid overheating the heating element)*)	
IF bError=FALSE THEN
	IF IOs.IO_Out_Vent_Camara=TRUE THEN
		Pcamara_Out(fIn:=fOut);
	ELSE
		Pcamara_Out(fIn:=0);
	END_IF
ELSE
	Pcamara_Out(fIn:=0);
	(*Escrever o erro para a HMI*)
END_IF

END_PROGRAM

// ---- POUs/Temperature Controller/PCamara_Out.TcPOU
PROGRAM PCamara_Out

VAR_INPUT
	fIn								: FLOAT;	
END_VAR

VAR
	bInit							: BOOL	:= TRUE;
	FB_CTRL_LIMIT : FB_CTRL_LIMITER;
	stParams     	: ST_CTRL_LIMITER_PARAMS;
	eMode			: E_CTRL_MODE;
	Init			: BOOL	:= TRUE;
	fOut			: FLOAT;
	eErrorId		: E_CTRL_ERRORCODES;
	bError 			: BOOL;
	
	aux 			: LREAL;

END_VAR

IF bInit THEN
	(* Init parameter struct *)
	stParams.tCtrlCycleTime   := T#10MS; 
  	stParams.tTaskCycleTime   := T#10MS; 
  	stParams.fMinOutput       :=0;
  	stParams.fMaxOutput       :=32767;

	(* ACTIVE --> normal operation *)
	eMode									:= eCTRL_MODE_ACTIVE;

	(* Reset the init flag *)
	bInit									:= FALSE;
END_IF

	(* Call function block *)
IF IOS.Temp_Camara_in>=17500 THEN
	aux:=0;
ELSE
	FB_CTRL_LIMIT(
		fIn:= (32767*fIn)/100, 
		fOut=>aux, 
		bMinLimit=>, 
		bMaxLimit=>, 
		eErrorId=>eErrorId , 
		bError=>bError, 
		stParams:=stParams );
END_IF

	(* Output sign   *)
IOS.A_Out_Aque_Ar:=LREAL_TO_UINT(aux);

END_PROGRAM

// ---- POUs/HMI/SetHMIVariables.TcPOU
PROGRAM SetHMIVariables
VAR
END_VAR

GVL.Temp_Camara_in := IOs.Temp_Camara_in;
GVL.Temp_8 := IOs.Temp_8;
GVL.Temp_Cabos := IOs.Temp_Cabos;
GVL.Temp_Chiller := IOs.Temp_Chiller;
GVL.Temp_Extrusor_1 := IOs.Temp_Extrusor_1;
GVL.Temp_Quadro := IOs.Temp_Quadro;
GVL.Temp_Tabuleiro := IOs.Temp_Tabuleiro;
IOs.IO_Out_Aque_Mesa := GVL.gvl_aquecimento_mesa;
IOs.IO_Out_Aque_Extrusor := GVL.gvl_aquecimento_extrusor;

END_PROGRAM

// ---- POUs/CNC/F2_Operation Mode/MM_TEst.TcPOU
FUNCTION_BLOCK HLI_ChannelModeManual2
VAR_INPUT

	stManualModeParameter 			: ST_ManualModeParameter;
	stManualModeControlElements 	: ST_ManualModeControlElements;

	bMMHMI				: BOOL;			(* static signal, for Manual Mode from HMI *)
	bReset				: BOOL;

END_VAR
VAR_OUTPUT
	bInManualMode		: BOOL;
	arrAxisInG201		: ARRAY[1..9] OF UINT;
	Busy				: BOOL;
	Err					: BOOL;
	nErrorState			: UINT;
	stManualModeState	: St_ManualModeState;
END_VAR
VAR
    nHliChIfcIdx		: INT;      (* Index of channel specific HLI area *)
	nState				: INT;
	pString				: POINTER TO STRING;

	pUnit				: POINTER TO MC_CONTROL_MCM_MODE_STATE_UNIT;
	pCommand			: POINTER TO HLI_PROC_TRANS_TO_MODE_STATE;

	pKey				: POINTER TO MC_CONTROL_HB_KEY_UNIT;
	pIncr				: POINTER TO MC_CONTROL_HB_TIP_PARAM_UNIT;

	stManualModeParameterOld : 	ST_ManualModeParameter;
	incOld				: UINT;
	nManualTypOld		: UINT;
	i					: UINT;
	bManual 			: BOOL;


	(* FBs for manual mode *)
	ManualActivation	: HLI_ManualActivation;

	(* Es können Global 9 Control Units verwendet werden, dies ist von ISG so vorgegeben *)
	ManualExecution				: ARRAY[1..9] OF HLI_ManualExecution;
	ManualExecutionRapidMode	: ARRAY[1..9] OF HLI_ManualExecutionRapidMode;

	ManualDeact			: HLI_ManualDeactivation;

	RTRapidKey			: R_TRIG;
	FTRapidKey			: F_TRIG;
	ActChannelModeOld 	: UDINT;
	TON_ModeChange		: TON;
	TON_TimeOut			: TON;

	ErrorState			: INT;
	nChan				: UINT;
	j					: INT;

	nCheckDeactivation	: UINT;
	strInitParameterOld	: STRING;

END_VAR

(* ========================================================= 	*)
(*     FB: HLI_ChannelModeManual2                            	*)
(* --------------------------------------------------------- 	*)
(*   Desc: Switch to Manual Mode and parametrize             	*)
(*   Author: TV                                         		*)
(*   Date: 18.07.2002                                        	*)
(*   Last: 13.12.2010                                        	*)
(*   Rev.: 4.0	                                              	*)
(* ========================================================= 	*)



nChan        := stManualModeParameter.stChannelParameter.nChan;
nHliChIfcIdx := stManualModeParameter.stChannelParameter.nChan - 1;

IF  nChan <= 0 OR gNrCh < nChan OR					(* check for channel no *)
	nChan > 2 THEN		(* check for zero pointer *)
	Busy := FALSE;
	RETURN; (* A b b r u c h *)
END_IF

IF  gpCh[nHliChIfcIdx] = 0 THEN		(* check for zero pointer *)
	Busy := FALSE;
	RETURN; (* A b b r u c h *)
END_IF


IF bMMHMI THEN
	Busy := FALSE;
	RETURN; (* A b b r u c h *)
END_IF


(* Handrad :

dem Kern IMMER die aktuellen Incremente mitteilen 
Hinweis : es können 6 Handräder verwendet werden
Siehe auch Handradparameter im SystemManager 
hr_data[0].adr_hr_zaehler                             0x0       
# Handradzaehleradresse (bei HW) bzw Index im HLI-Array
*)


(* Vorgabe der Handrad Inkremente, es werden bis zu 6 Handräder unterstützt *)
FOR j := 1 TO (HLI_HW_MAXIDX + 1) DO
	gpCh[nHliChIfcIdx]^.hb_mc_control.handwheel_incs[j-1].enable_w  := TRUE;
	gpCh[nHliChIfcIdx]^.hb_mc_control.handwheel_incs[j-1].command_w := stManualModeControlElements.nHandwheelInc[j];
END_FOR

IF 	CNCSystem.Channel[nChan].ActMode <> HLI_IMCM_MANUAL_MODE AND
	CNCSystem.Channel[nChan].ActMode <> HLI_IMCM_AUTOMATIC_MODE   AND
	CNCSystem.Channel[nChan].ActMode <> HLI_IMCM_MDI_MODE THEN
		strInitParameterOld := '';
		Busy := FALSE;
		nState := 0;
	RETURN; (* A b b r u c h *)
ELSE
	bManual := TRUE;
END_IF


IF  CNCSystem.Channel[nChan].ActMode <> HLI_IMCM_MANUAL_MODE THEN
	strInitParameterOld := '';
END_IF


(* Clear all request from the HMI *)
IF gpCh[nHliChIfcIdx]^.hb_mc_control.key[0].request_semaphor_rw THEN
	gpCh[nHliChIfcIdx]^.hb_mc_control.key[0].request_semaphor_rw := FALSE;
END_IF

IF gpCh[nHliChIfcIdx]^.hb_mc_control.activation.request_semaphor_rw THEN
	gpCh[nHliChIfcIdx]^.hb_mc_control.activation.request_semaphor_rw := FALSE;
END_IF

IF gpCh[nHliChIfcIdx]^.hb_mc_control.tip_parameter.request_semaphor_rw THEN
	gpCh[nHliChIfcIdx]^.hb_mc_control.tip_parameter.request_semaphor_rw := FALSE;
END_IF

IF gpCh[nHliChIfcIdx]^.hb_mc_control.jog_parameter.request_semaphor_rw THEN
	gpCh[nHliChIfcIdx]^.hb_mc_control.jog_parameter.request_semaphor_rw := FALSE;
END_IF


Busy := TRUE;

IF bReset THEN
	nState := 0;
	nErrorState := 0;
	Err := FALSE;
	bInManualMode := FALSE;
END_IF


IF stManualModeParameter.stChannelParameter.nManualTyp = 4 THEN

	PRG_AnalogJoystick(	nLogAxisNr:= stManualModeParameter.stAxisParameter.stControlUnit[1].nLogAxisNumber,
								Analog_Value:= stManualModeControlElements.stControlJoystickValue[1],
								AnalogValueMin:= stManualModeParameter.stJoystickParameter.AnalogValueMin,
								AnalogValueMax:= stManualModeParameter.stJoystickParameter.AnalogValueMax,
								AnalogValueZeroDeadBand:= stManualModeParameter.stJoystickParameter.AnalogValueZeroDeadBand,
								bKeyPos:= stManualModeControlElements.stControlKeys[1].bKeyPos,
								bKeyNeg:= stManualModeControlElements.stControlKeys[1].bKeyNeg);

	PRG_AnalogJoystick(	nLogAxisNr:= stManualModeParameter.stAxisParameter.stControlUnit[2].nLogAxisNumber,
								Analog_Value:= stManualModeControlElements.stControlJoystickValue[2],
								AnalogValueMin:= stManualModeParameter.stJoystickParameter.AnalogValueMin,
								AnalogValueMax:= stManualModeParameter.stJoystickParameter.AnalogValueMax,
								AnalogValueZeroDeadBand:= stManualModeParameter.stJoystickParameter.AnalogValueZeroDeadBand,
								bKeyPos:= stManualModeControlElements.stControlKeys[2].bKeyPos,
								bKeyNeg:= stManualModeControlElements.stControlKeys[2].bKeyNeg);

	PRG_AnalogJoystick(	nLogAxisNr:= stManualModeParameter.stAxisParameter.stControlUnit[3].nLogAxisNumber,
								Analog_Value:= stManualModeControlElements.stControlJoystickValue[3],
								AnalogValueMin:= stManualModeParameter.stJoystickParameter.AnalogValueMin,
								AnalogValueMax:= stManualModeParameter.stJoystickParameter.AnalogValueMax,
								AnalogValueZeroDeadBand:= stManualModeParameter.stJoystickParameter.AnalogValueZeroDeadBand,
								bKeyPos:= stManualModeControlElements.stControlKeys[3].bKeyPos,
								bKeyNeg:= stManualModeControlElements.stControlKeys[3].bKeyNeg);

	PRG_AnalogJoystick(	nLogAxisNr:= stManualModeParameter.stAxisParameter.stControlUnit[4].nLogAxisNumber,
								Analog_Value:= stManualModeControlElements.stControlJoystickValue[4],
								AnalogValueMin:= stManualModeParameter.stJoystickParameter.AnalogValueMin,
								AnalogValueMax:= stManualModeParameter.stJoystickParameter.AnalogValueMax,
								AnalogValueZeroDeadBand:= stManualModeParameter.stJoystickParameter.AnalogValueZeroDeadBand,
								bKeyPos:= stManualModeControlElements.stControlKeys[4].bKeyPos,
								bKeyNeg:= stManualModeControlElements.stControlKeys[4].bKeyNeg);

	PRG_AnalogJoystick(	nLogAxisNr:= stManualModeParameter.stAxisParameter.stControlUnit[5].nLogAxisNumber,
								Analog_Value:= stManualModeControlElements.stControlJoystickValue[5],
								AnalogValueMin:= stManualModeParameter.stJoystickParameter.AnalogValueMin,
								AnalogValueMax:= stManualModeParameter.stJoystickParameter.AnalogValueMax,
								AnalogValueZeroDeadBand:= stManualModeParameter.stJoystickParameter.AnalogValueZeroDeadBand,
								bKeyPos:= stManualModeControlElements.stControlKeys[5].bKeyPos,
								bKeyNeg:= stManualModeControlElements.stControlKeys[5].bKeyNeg);

ELSE
	(* Achsoverride wieder auf 100 % setzen *)
	FOR j := 1 TO UDINT_TO_INT(stManualModeParameter.stChannelParameter.nControlUnits) DO
		HLI_SetAxisOverride(nAxisNr := stManualModeParameter.stAxisParameter.stControlUnit[j].nLogAxisNumber, nOverride := 1000);
	END_FOR
END_IF

(******** Parallelinterpolation mit G201 *************************************)
IF CNCSystem.Channel[nChan].ActMode = HLI_IMCM_AUTOMATIC_MODE OR CNCSystem.Channel[nChan].ActMode = HLI_IMCM_MDI_MODE THEN
	arrAxisInG201 := HLI_AxisInManualMode(nChan);
	FOR j := 1 TO UDINT_TO_INT(stManualModeParameter.stChannelParameter.nControlUnits) DO
		stManualModeParameter.stAxisParameter.stControlUnit[j].nLogAxisNumber := arrAxisInG201[j];
	END_FOR
ELSE
	FOR j := 1 TO UDINT_TO_INT(stManualModeParameter.stChannelParameter.nControlUnits) DO
	arrAxisInG201[j] := 0;
	END_FOR
END_IF
(* **************************************************************************** *)




CASE nState OF


	0: (* IDLE *)
		Busy := FALSE;
		bInManualMode := FALSE;


		IF (CNCSystem.Channel[nChan].ActMode = HLI_IMCM_MANUAL_MODE AND stManualModeParameter.stChannelParameter.nManualTyp <> 0 AND CNCSystem.Channel[nChan].ActState = HLI_IMCM_PROCESS_ACTIVE) OR (* Manual Mode *)
			(arrAxisinG201[1] <> 0)	 (* mindestens eine Achse in G201 *) AND
			(CNCSystem.Channel[nChan].ActState = HLI_IMCM_PROCESS_ACTIVE) (* Channel is active *)
		THEN

			nErrorState := 0;
			Err := FALSE;


			stManualModeParameterOld	:= stManualModeParameter;
			ActChannelModeOld			:= cncsystem.Channel[nChan].ActMode;
			TON_ModeChange(in:=FALSE);
			i:= 1;
			nState := 10;

		END_IF


		(* Evt. hier die Betriebsart auf Standby und danach
		wieder in Manual umschalten *)



	10:

			(* Beim Mode change wird eine Verzoegerung benötigt, weil
				die TcApplication bei Anwahl des Manual Mode den Handbetrieb 
				ebenfalls parametriert 
			 *)
			ManualDeact(bExecute := FALSE);
			TON_ModeChange(in:=TRUE, PT:=T#30ms);

			IF TON_ModeChange.Q THEN
				TON_ModeChange(in:=FALSE);
				i :=1;
				nCheckDeactivation := 0;
				nState := 20;
			END_IF



	20: (* deselecting axis first *)
		IF gpCh[nHliChIfcIdx]^.bahn_state.coord_r[i-1].log_achs_nr_r <> 0 THEN
			nCheckDeactivation := nCheckDeactivation + 1;

			ManualDeact(nChan := nChan, nAxisIndex :=i, bExecute := TRUE);

			IF ManualDeact.Busy THEN
				nState := 25;
			END_IF
		ELSE
			IF nCheckDeactivation < gNrAx THEN
				i := i+1;

				IF i > HLI_CH_AX_MAX THEN
					i := 1;
					nState := 26;
				END_IF

			ELSE
				ManualActivation(bExecute := FALSE);
				i := 1;
				nState := 26;
			END_IF
		END_IF




	25:
		ManualDeact(bExecute := FALSE);

		IF ManualDeact.Err THEN
			Err := TRUE;
			nErrorState := nState;
			nState := 99;
		END_IF

		IF ManualDeact.Busy = FALSE THEN

			IF i >= HLI_CH_AX_MAX AND i <> 0  THEN
				i:=1; (* reset the array counter *)
				ManualActivation(bExecute := FALSE);
				i := 1;
				nState := 26;
			ELSE
				ManualDeact(bExecute := FALSE);
				nState := 20;
				i:= i+1;
			END_IF
		END_IF

		(* Activation of an manual mode string, eg. TRAFO ON or ECS ON *)
26:		IF (stManualModeParameter.stChannelParameter.strInitParameter  <> '' AND stManualModeParameter.stChannelParameter.strInitParameter <> strInitParameterOld) THEN

			gpCh[nHliChIfcIdx]^.channel_mc_control.mode_and_state.command_w.to_mode := HLI_IMCM_MANUAL_MODE ;
			gpCh[nHliChIfcIdx]^.channel_mc_control.mode_and_state.command_w.to_state := HLI_IMCM_PROCESS_SELECTED;
			gpCh[nHliChIfcIdx]^.channel_mc_control.mode_and_state.command_w.channel_number := nChan;
			pString := ADR(gpCh[nHliChIfcIdx]^.channel_mc_control.mode_and_state.command_w.parameter);
			pString^ := '';

			gpCh[nHliChIfcIdx]^.channel_mc_control.mode_and_state.command_semaphor_rw := TRUE;
			TON_TimeOut(in:= FALSE);
			nState := 27;

		ELSE
			nState := 30;
		END_IF


27:		IF (gpCh[nHliChIfcIdx]^.channel_mc_control.mode_and_state.command_semaphor_rw = FALSE) THEN


			gpCh[nHliChIfcIdx]^.channel_mc_control.mode_and_state.command_w.to_mode := HLI_IMCM_MANUAL_MODE ;
			gpCh[nHliChIfcIdx]^.channel_mc_control.mode_and_state.command_w.to_state := HLI_IMCM_PROCESS_ACTIVE;
			gpCh[nHliChIfcIdx]^.channel_mc_control.mode_and_state.command_w.channel_number := nChan;
			pString := ADR(gpCh[nHliChIfcIdx]^.channel_mc_control.mode_and_state.command_w.parameter);
			pString^ := stManualModeParameter.stChannelParameter.strInitParameter;

			gpCh[nHliChIfcIdx]^.channel_mc_control.mode_and_state.command_semaphor_rw := TRUE;
			TON_ModeChange(in:=FALSE);
			TON_TimeOut(in:= FALSE);
			nState := 28;
		END_IF

		TON_TimeOut(in:=TRUE, PT:=T#5s);
		IF TON_TimeOut.Q THEN
			nState := 99;
		END_IF

28:		IF (gpCh[nHliChIfcIdx]^.channel_mc_control.mode_and_state.command_semaphor_rw = FALSE) THEN
			TON_ModeChange(in:=TRUE, PT:=T#1s);
			IF  TON_ModeChange.Q THEN
				strInitParameterOld := stManualModeParameter.stChannelParameter.strInitParameter;
				nState := 30;
			END_IF
		END_IF

		TON_TimeOut(in:=TRUE, PT:=T#5s);
		IF TON_TimeOut.Q THEN
			nState := 99;
		END_IF

30: 	(* --- activate KeyControlUnit 1 - 4 --- *)

			ManualActivation(bExecute := TRUE,
										nChan := nChan,
										nManualTyp 		:= stManualModeParameter.stChannelParameter.nManualTyp,
										nKeyControlUnit := i + stManualModeParameter.stChannelParameter.nControlUnits * (nHliChIfcIdx),
										nHBA_Res 		:= stManualModeParameter.stChannelParameter.nHandwheelResolution,
										Inc 			:= stManualModeParameter.stChannelParameter.nInc,
										Speed 			:= stManualModeParameter.stAxisParameter.stControlUnit[i].nSpeed,
										nLogAxisNr 		:= stManualModeParameter.stAxisParameter.stControlUnit[i].nLogAxisNumber);
			nState := 35;

35: 	(* waiting for acknowledge *)

		ManualActivation(bExecute := FALSE);

		IF ManualActivation.Err THEN
			Err := TRUE;
			nErrorState := nState;
			nState := 99;
		END_IF

		IF ManualActivation.Busy = FALSE THEN

			IF i >= stManualModeParameter.stChannelParameter.nControlUnits THEN
				i:=1; (* reset the array counter *)
				ManualActivation(bExecute := FALSE);
				i := 1;
				nState := 40;
			ELSE
				ManualActivation(bExecute := FALSE);
				nState := 30;
				i:= i+1;
			END_IF
		END_IF

	40: (* endlich Handbetrieb *)
		bInManualMode := TRUE;

		FOR j := 1 TO UDINT_TO_INT(stManualModeParameter.stChannelParameter.nControlUnits) DO
			ManualExecution[j](	nChan := nChan,
								nKeyControlUnit := j + stManualModeParameter.stChannelParameter.nControlUnits * (nHliChIfcIdx),
								bKeyPos := stManualModeControlElements.stControlKeys[j].bKeyPos,
								bKeyNeg := stManualModeControlElements.stControlKeys[j].bKeyNeg); (* no timeouts *)

			ManualExecutionRapidMode[j](nChan := nChan,
										nKeyControlUnit := j + stManualModeParameter.stChannelParameter.nControlUnits * (nHliChIfcIdx),
										bExecute := stManualModeControlElements.stControlKeys[j].bKeyRapid); (* no timeouts *)


		END_FOR

		(* end of manual mode *)
		IF (bManual = FALSE) OR
				MEMCMP(ADR(stManualModeParameter),ADR(stManualModeParameterOld),SIZEOF(stManualModeParameter))<>0 OR
				cncsystem.Channel[nChan].ActMode <> ActChannelModeOld OR
				stManualModeParameter.stChannelParameter.nManualTyp = 0
			THEN

			FOR j := 1 TO UDINT_TO_INT(stManualModeParameter.stChannelParameter.nControlUnits) DO
				ManualExecution[j](nChan := nChan,	nKeyControlUnit := j + stManualModeParameter.stChannelParameter.nControlUnits * (nHliChIfcIdx), bKeyPos := FALSE, bKeyNeg := FALSE); (* no timeouts *)
			END_FOR


			i:=1 (* resets the counter for the following deactivation *);
			ManualDeact(bExecute := FALSE);

			stManualModeParameterOld 	:= stManualModeParameter;

			IF cncsystem.Channel[nChan].ActMode <> ActChannelModeOld OR stManualModeParameter.stChannelParameter.nManualTyp = 0 THEN
				ActChannelModeOld := cncsystem.Channel[nChan].ActMode;
				TON_ModeChange(in:=FALSE);
				nState := 0;
			ELSE
				nState := 0; (* evt. wird hier auch eine Verzoegerungszeit benötigt,
									  Fehler 150054 dann nState = 0 *)
				bInManualMode := FALSE;
			END_IF
		END_IF


	99: (* error handling *)
		ErrorState := nState;
		(* end of manual mode *)
		IF bManual = FALSE THEN
			Busy := FALSE;
			nState := 1;
		END_IF


END_CASE

END_FUNCTION_BLOCK

// ---- POUs/CNC/F3_Control/HLI_ChannelGetActiveFeed.TcPOU
FUNCTION HLI_ChannelGetActiveFeed : LREAL
VAR_INPUT
	nChan					: UINT;			(* Number of channel *)
END_VAR
VAR
	nHliChIdx			: UINT;
END_VAR

(* ========================================================= *)
(*    FUN: HLI_ChannelGetActiveFeed                          *)
(* --------------------------------------------------------- *)
(*   Desc: Active feed                                       *)
(* Return: Active feed of the channel during interpolation   *)
(* Author: MK                                                *)
(*   Date: 30.11.2015                                        *)
(*   Rev.: 1.0                                               *)
(* ========================================================= *)


nHliChIdx := nChan - 1;

IF nChan <= 0 OR gNrCh < nChan OR			(* check for channel no *)
	gpCh[nHliChIdx] = 0 THEN					(* check for zero pointer *)
	HLI_ChannelGetActiveFeed := 0.0;
	RETURN; (* e x i t *)
END_IF


HLI_ChannelGetActiveFeed := DINT_TO_LREAL(gpCh[nHliChIdx]^.bahn_state.active_feed_r) * (60.0/1000000.0);

END_FUNCTION

// ---- POUs/CNC/F3_Control/HLI_ChannelSetHandWheelIncs.TcPOU
FUNCTION HLI_ChannelSetHandWheelIncs : bool
VAR_INPUT
	nChan					: UINT;			(* Number of channel *)
	nIncs					: DINT;			(* Number of increments *)
	nHandWheel			: INT;			(* Number of the handwheel *)
END_VAR
VAR
	nHliChIdx			: UINT;
END_VAR

(* ========================================================= *)
(*    FUN: HLI_ChannelSetHandWheelIncs                       *)
(* --------------------------------------------------------- *)
(*   Desc:                                                   *)
(* Author: MK                                                *)
(*   Date: 21.12.2011                                        *)
(*   Rev.: 1.0                                               *)
(* ========================================================= *)


nHliChIdx := nChan - 1;

IF nChan <= 0 OR gNrCh < nChan OR			(* check for channel no *)
	gpCh[nHliChIdx] = 0 THEN					(* check for zero pointer *)
	HLI_ChannelSetHandWheelIncs := FALSE;
	RETURN; (* e x i t *)
END_IF

// MK check
// todo check for handwheel nr

gpCh[nHliChIdx]^.hb_mc_control.handwheel_incs[nHandWheel].command_w := nIncs;

HLI_ChannelSetHandWheelIncs := TRUE;

END_FUNCTION

// ---- POUs/CNC/F9_Misc/Security/CheckCNCAlive.TcPOU
FUNCTION CheckCncAlive : INT
VAR_INPUT
	nChan					: UINT;			(* Number of channel *)
END_VAR
VAR
	nHliChIdx			: UINT;
END_VAR

(* The assumption is made that the cycle time of the PLC is at least twice as big as the CNC cycle time.

The Cycle time of CNC is displayed in element:
	gpCh[0]^.head.lc_watchdog.cycle_time_r

remark: Take care if PLC cycle is smaller not to check CNC faster as possible !!!

To simulate failure of CNC set cycle time of PLC smaller than CNC (Resource/task configuration).
*)

nHliChIdx := nChan - 1;

IF nChan <= 0 OR gNrCh < nChan OR			(* check for channel no *)
	gpCh[nHliChIdx] = 0 THEN					(* check for zero pointer *)
	CheckCncAlive := -1;
	RETURN; (* e x i t *)
END_IF

(* Copy current state of live sign to watchdog state *)
gpCh[nHliChIdx]^.head.lc_watchdog.alive_state_w := gpCh[nHliChIdx]^.head.lc_watchdog.alive_rw;

IF gpCh[nHliChIdx]^.head.lc_watchdog.alive_rw THEN
	CheckCncAlive := 1;	(* CNC alive *)
ELSE
	CheckCncAlive := 0;	(* CNC not alive *)
END_IF 

(* reset live sign for next cycle *)
gpCh[nHliChIdx]^.head.lc_watchdog.alive_rw	:= FALSE;

END_FUNCTION

// ---- POUs/CNC/F9_Misc/Security/SetPlcAlive.TcPOU
FUNCTION SetPlcAlive : BOOL
VAR_INPUT
	nChan					: UINT;			(* Number of channel *)
END_VAR
VAR
	nHliChIdx			: UINT;
END_VAR

(*
Display PLC is just alive (Trigger Watchdog to MC)
If PLC is stopped here, alive sign is missing.
-> CNC raises error message
-> CNC stops movement with internal FEEDHOLD
-> system has to be restarted (after removal of error)
*)

nHliChIdx := nChan - 1;

IF nChan <= 0 OR gNrCh < nChan OR			(* check for channel no *)
	gpCh[nHliChIdx] = 0 THEN					(* check for zero pointer *)
	SetPlcAlive := FALSE;
	RETURN; (* e x i t *)
END_IF

gpCh[nHliChIdx]^.head.mc_watchdog.alive_rw := TRUE;

SetPLCAlive	:= TRUE;

END_FUNCTION

// ---- POUs/General/Examples.TcPOU
PROGRAM Examples
VAR
	pAxis								: POINTER TO HIGH_LEVEL_INTERFACE_AX;
	pChannel							: POINTER TO HIGH_LEVEL_INTERFACE_CH;
	cmdValue							: DINT;
	cmdRev							: DINT;

(*
	DevInfo							: ADSRDDEVINFO;
	rdInfo							: BOOL;
*)

	fbFileOffset					: FB_ReadFileOffset;
	start								: BOOL;
	fileOffset						: DINT;

	fbFileName						: FB_ReadFileName;
	fileName							: STRING(255);
	showMsg							: BOOL := TRUE;

	fbPParamValue					: FB_ReadPParamValue;
	startReadValue 				: BOOL;
	pparamName						: STRING;
	pparamValue						: LREAL;
	
	
END_VAR


(* shows how to get the data of the first axis *)
pAxis := gpAx[0];

(* shows how to get the data of the first channel *)
pChannel := gpCh[0];

(* External commanding of an axis *)
pAxis^.lr_mc_control.add_cmd_values.command_w := cmdValue;

(* Commanded revolution of the first (spindle) axis *)
cmdRev := pAxis^.lr_state.cmd_rev_r;

(* Reads the device info *)
(*
DevInfo(NETID:='', PORT:=10000, RDINFO:=rdInfo, TMOUT:=T#2s); 
*)



(* ----------------------------------------------
	Shows how to read GEO task exceed counter
   ---------------------------------------------- *)
(*readGeoTaskExceedCounter(bStart:=bStartGTEC, pDest:=ADR(exCounter)); *)


(* ----------------------------------------------
	Shows how to read file offset and file name
   ---------------------------------------------- *)
(*fbFileOffset(nIdxGrp:=16#20100 + 1, bStart:=start, pDest:=ADR(fileOffset));
fbFileName(nIdxGrp:=16#20100 + 1, bStart:=start, pDest:=ADR(fileName)); *)


(* ----------------------------------------------
	Shows how to read P-Parameter value
   ---------------------------------------------- *)
(* pparamName := 'P5'; *)
(*
IF startReadValue = TRUE THEN
	fbPParamValue(
				nIdxGrp := 16#22301,
				bStart := startReadValue,
				pSrc := ADR(pparamName),
				pDest := ADR(pparamValue));
	IF fbPParamValue.Busy = FALSE THEN
		startReadValue := FALSE;
	END_IF
END_IF
*)


(* ----------------------------------------------
	Shows how to read the current axis position
   ---------------------------------------------- *)

END_PROGRAM

// ---- POUs/General/FB_ReadPParamValue.TcPOU
FUNCTION_BLOCK FB_ReadPParamValue
VAR_INPUT
   nIdxGrp              : UDINT;
   bStart               : BOOL;
   pSrc                 : POINTER TO STRING;
   pDest                : POINTER TO DINT;
END_VAR
VAR_OUTPUT
   Busy                 : BOOL;
   bErr                 : BOOL;
   bErrID               : UDINT;
END_VAR
VAR
   fbAdsRWEx            : ADSRDWRTEX;
   bStarted             : BOOL;
END_VAR

(* ========================================================= *)
(*     FB: FB_ReadFileOffset                                 *)
(* --------------------------------------------------------- *)
(*   Desc: Example, shows how to read file name              *)
(*       : from the CNC                                      *)
(* Author: MK                                                *)
(*   Date: 21.12.2011                                        *)
(*   Rev.: 1.0                                               *)
(* ========================================================= *)


IF bStarted = FALSE THEN
   IF bStart = TRUE THEN
      bStarted := TRUE;
      bErr := FALSE;
      Busy := TRUE;
   END_IF
END_IF

IF bStarted THEN
   (* raising edge of Timer triggers read/write request *)

	fbAdsRWEx(NetID := '', Port := 552, IdxGrp := nIdxGrp, IdxOffs := 16#01C,
				WRITELEN := 2, READLEN := 8, SRCADDR := pSrc, DESTADDR := pDest, WRTRD := bStarted, TMOUT := T#2s);
   IF NOT fbAdsRWEx.Busy THEN
      (* There was an error in the execution of the read/write request *)
      IF fbAdsRWEx.Err THEN
         bErr := TRUE;
      END_IF
		bErrID := fbAdsRWEx.ERRID;
      fbAdsRWEx(WRTRD := FALSE);
      bStarted := FALSE;
      Busy := FALSE;
   END_IF
END_IF

END_FUNCTION_BLOCK

// ---- POUs/General/FB_AdsRead.TcPOU
FUNCTION_BLOCK FB_AdsRead
VAR_INPUT
   sNetId               : T_AmsNetId;
	nPort                : T_AmsPort;
   nIdxGrp              : UDINT;
   nIdxOffs             : UDINT;
	nLen						: UDINT;
   bStart               : BOOL;
   pDest                : POINTER TO PVOID;
END_VAR
VAR_OUTPUT
   bBusy                : BOOL;
   bErr                 : BOOL;
END_VAR
VAR
   fbRead               : ADSREAD;
   bStarted             : BOOL;
END_VAR

(* ========================================================= *)
(*     FB: FB_AdsRead                                        *)
(* --------------------------------------------------------- *)
(*   Desc: Ads Read                                          *)
(* Author: MK                                                *)
(*   Date: 21.12.2011                                        *)
(*   Rev.: 1.0                                               *)
(* ========================================================= *)


IF bStart = TRUE AND bStarted = FALSE THEN
	bStarted := TRUE;
	bErr := FALSE;
	bBusy := TRUE;
END_IF

IF bStarted THEN
   fbRead(NetID:=sNetId, Port:=nPort, IdxGrp:=nIdxGrp, IdxOffs:=nIdxOffs,
         LEN:=nLen, DestAddr:=pDest, READ:=bStarted, TMOUT:=T#3S);
   IF NOT fbRead.Busy THEN
      IF fbRead.Err THEN
         bErr := TRUE;
      END_IF
      fbRead(READ := FALSE);
      bStarted := FALSE;
      bBusy := FALSE;
   END_IF
END_IF

END_FUNCTION_BLOCK

// ---- POUs/HMI/DIntToString.TcPOU
FUNCTION DIntToString : STRING
VAR_INPUT
	val					: DINT;
END_VAR
VAR
	v1						: INT;
	v2						: dINT;
	valString			: STRING;
END_VAR

IF val >= 0 THEN
	val := val + 5;
ELSE
	val := val - 5;
END_IF

v1 := LREAL_TO_INT(TRUNC(val/10000));
v2 := ABS(val MOD 10000)/10;

IF v1 = 0 AND val < 0 THEN
	valString := '-0';
ELSE
	valString := INT_TO_STRING(v1);
END_IF

IF v2 >= 100 THEN
	valString := CONCAT(str1 := valString, str2 := '.');
ELSIF v2 >= 10 THEN
	valString := CONCAT(str1 := valString, str2 := '.0');
ELSE
	valString := CONCAT(str1 := valString, str2 := '.00');
END_IF

valString := CONCAT(str1 := valString, str2 := DINT_TO_STRING(v2));

DIntToString := valString;

END_FUNCTION

// ---- POUs/HMI/LRealToString.TcPOU
FUNCTION LRealToString : STRING
VAR_INPUT
	val					: LREAL;
END_VAR
VAR
	v1						: INT;
	v2						: INT;
	valString			: STRING;
END_VAR

v1 := LREAL_TO_INT(TRUNC(val));
v2 := ABS(LREAL_TO_INT((val - v1)*1000));

IF v1 = 0 AND val < 0 THEN
	valString := '-0';
ELSE
	valString := INT_TO_STRING(v1);
END_IF

IF v2 >= 100 THEN
	valString := CONCAT(str1 := valString, str2 := '.');
ELSIF v2 >= 10 THEN
	valString := CONCAT(str1 := valString, str2 := '.0');
ELSE
	valString := CONCAT(str1 := valString, str2 := '.00');
END_IF

valString := CONCAT(str1 := valString, str2 := INT_TO_STRING(v2));

LRealToString := valString;

END_FUNCTION
